PROGRAM MAIN
VAR
END_VAR

END_PROGRAM

(* stored: Version 1.1.0.1
   POU MAIN: Id {f9a225d6-227e-4846-a38a-e189c9e25045} *)
